# EPICS substitutions: db/ecmcEL6080.substitutions
# All fields related to postion scaling and alarms
file ecmcEcSlave.template
{
    pattern {}
            {}
}

file ecmcEL6080.template
{
    pattern {}
            {}
}

file ecmcEL6080_app.template
{
    pattern {}
            {}
}
